// TIA Portal V20 export
TYPE "UDT_MTP_LockView4"
// Interface Definition LockView4
   STRUCT
      WQC { ExternalWritable := 'False'} : Byte := 16#FF;   // Worst Quality Code variable
      Logic { ExternalWritable := 'False'} : Bool;   // Logical behaviour, false: OR, true: AND
      In1En { ExternalWritable := 'False'} : Bool;   // Locking Input 1 - Enable, 0: Input not used, 1: Input is used
      In1 { ExternalWritable := 'False'} : Bool;   // Locking Input 1 - Value
      In1QC { ExternalWritable := 'False'} : Byte := 16#FF;   // Locking Input 1 - Quality Code
      In1Inv { ExternalWritable := 'False'} : Bool;   // Locking Input 1 - Inversion Enable, 0: Input not inverted, 1: Input inverted
      In1Txt { ExternalWritable := 'False'} : String[16] := '';   // Locking Input 1 - Additional Text
      In2En { ExternalWritable := 'False'} : Bool;   // Locking Input 2 - Enable, 0: Input not used, 1: Input is used
      In2 { ExternalWritable := 'False'} : Bool;   // Locking Input 2 - Value
      In2QC { ExternalWritable := 'False'} : Byte := 16#FF;   // Locking Input 2 - Quality Code
      In2Inv { ExternalWritable := 'False'} : Bool;   // Locking Input 2 - Inversion Enable, 0: Input not inverted, 1: Input inverted
      In2Txt { ExternalWritable := 'False'} : String[16] := '';   // Locking Input 2 - Additional Text
      In3En { ExternalWritable := 'False'} : Bool;   // Locking Input 3 - Enable, 0: Input not used, 1: Input is used
      In3 { ExternalWritable := 'False'} : Bool;   // Locking Input 3 - Value
      In3QC { ExternalWritable := 'False'} : Byte := 16#FF;   // Locking Input 3 - Quality Code
      In3Inv { ExternalWritable := 'False'} : Bool;   // Locking Input 3 - Inversion Enable, 0: Input not inverted, 1: Input inverted
      In3Txt { ExternalWritable := 'False'} : String[16] := '';   // Locking Input 3 - Additional Text
      In4En { ExternalWritable := 'False'} : Bool;   // Locking Input 4 - Enable, 0: Input not used, 1: Input is used
      In4 { ExternalWritable := 'False'} : Bool;   // Locking Input 4 - Value
      In4QC { ExternalWritable := 'False'} : Byte := 16#FF;   // Locking Input 4 - Quality Code
      In4Inv { ExternalWritable := 'False'} : Bool;   // Locking Input 4 - Inversion Enable, 0: Input not inverted, 1: Input inverted
      In4Txt { ExternalWritable := 'False'} : String[16] := '';   // Locking Input 4 - Additional Text
      Out { ExternalWritable := 'False'} : Bool;   // Locking Result Output
      OutQC { ExternalWritable := 'False'} : Byte := 16#FF;   // Locking Result Output - Quality Code
   END_STRUCT;
END_TYPE
